PROGRAM P_Demo_CEIL
VAR
    lrPackageWeightKg : LREAL := 0.3; // 称重模块的读数；在线写值模拟不同包裹重量
    lrChargeTier      : LREAL; // 向上取整后的收费档位（公斤）
    nChargeYuan       : DINT; // 收费系统接收的整数金额（元）
END_VAR

// =============================================================================
// 场景：分拣线按重量阶梯收费——0.01-1.00kg 收 1 元、1.01-2.00kg 收 2 元……
//       需要把称重模块的 LREAL 读数向上取整到下一公斤，得到收费档位。
//
// 价值：CEIL 一行替代多段 IF/ELSIF 阈值判断；返回 LREAL 还能处理超出 DINT
//       范围的大数（极少数大宗物料场景）；负数侧朝 +∞ 取整有明确语义。
//
// 验证步骤：
//   1. 引用 Tc2_Math
//   2. 在 PLC 项目右键 → Add Existing Item (.TcPOU) → 选本文件 → OK
//   3. 编译、登录、运行
//   4. 在线 monitor 看：
//      - lrPackageWeightKg = 0.3 → lrChargeTier 应为 1.0，nChargeYuan = 1
//      - 在线改 lrPackageWeightKg = 1.0 → lrChargeTier 仍 1.0（边界含值）
//      - 改 1.01 → 2.0
//      - 改 -0.3 → 0.0 （负数朝 +∞，验证 CEIL 不是绝对值变大）
// =============================================================================

// 单行调用：CEIL 朝 +∞ 方向取整，正数侧符合"向上取"直觉
lrChargeTier := CEIL(lrPackageWeightKg);

// LREAL → DINT 显式转换，规避隐式转换编译警告
// （CEIL 已保证 lrChargeTier 是整数值，转换不损失精度）
nChargeYuan := LREAL_TO_DINT(lrChargeTier);

END_PROGRAM

(* stored: Version 1.1.0.1, ProductVersion 3.1.4024.5
   POU P_Demo_CEIL: Id {19c034a9-1a17-573b-8aad-81ffb1e0f353}, SpecialFunc None *)
